FUNCTION_BLOCK ARM_COMM (* Peroidic event generator *)
  (* Standard: 61499-1 Annex A; Description: Copyright (c) 2017 fortiss GmbH This program and the accompanying materials are made available under the terms of the Eclipse Public License 2.0 which is available at https://www.eclipse.org/legal/epl-2.0/ SPDX-License-Identifier: EPL-2.0 *)
  (* Version 1.0, 2017-09-21, Alois Zoitl, fortiss GmbH, initial API and implementation and/or initial documentation *)
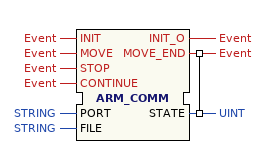
  EVENT_INPUT
    INIT;
    MOVE;
    STOP;
    CONTINUE;
  END_EVENT
  EVENT_OUTPUT
    INIT_O;
    MOVE_END WITH STATE;
  END_EVENT
  VAR_INPUT
    PORT : STRING;
    FILE : STRING;
  END_VAR
  VAR_OUTPUT
    STATE : UINT;
  END_VAR
END_FUNCTION_BLOCK
